SYSTEM Simple Test System
  (* Version 1.0, 2007-08-07, Goran Cengic, Chalmers *)
  DEVICE Test Device : DeviceType_not_used
    RESOURCE Test Resource : ResourceType_not_used
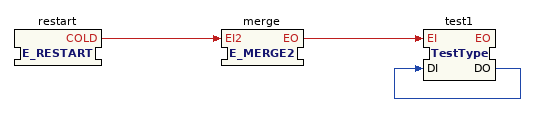
      FBS
        restart : E_RESTART;
        merge : E_MERGE2;
        test1 : TestType;
      END_FBS
      EVENT_CONNECTIONS
        restart.COLD TO merge.EI2;
        merge.EO TO test1.EI;
      END_CONNECTIONS
      DATA_CONNECTIONS
        test1.DO TO test1.DI;
      END_CONNECTIONS
    END_RESOURCE
  END_DEVICE
END_SYSTEM
(* other elements stored in the file *)
(* Connection Source="test1.EO" Destination="merge.EI1" / *)
